{attribute 'linkalways'} 
{attribute 'no_explicit_call' := 'This FB is a CLASS and must be accessed using methods or properties'}
{attribute 'enable_dynamic_creation'}
FUNCTION_BLOCK Node_F_VN_FillContainerExp_INT EXTENDS VisionNode
VAR
    ipContainer : _ITcVnContainer;
    nValue : _INT(0);
    nStartIdx : _ULINT(0);
    nCount : _ULINT(0);
    hrPrev : _HRESULT(S_OK);
    hresult : _HRESULT(S_OK);
END_VAR

METHOD PUBLIC  Clone : I_Node
VAR
    pNode : POINTER TO Node_F_VN_FillContainerExp_INT;
END_VAR
pNode := __NEW(Node_F_VN_FillContainerExp_INT);
Clone := pNode^;
END_METHOD

METHOD FB_init : BOOL
VAR_INPUT
    bInitRetains : BOOL; // if TRUE, the retain variables are initialized (warm start / cold start)
    bInCopyCode : BOOL;  // if TRUE, the instance afterwards gets moved into the copy code (online change)
END_VAR
AddInput('ipContainer', ipContainer);
AddParameter('nValue', nValue);
AddParameter('nStartIdx', nStartIdx);
AddParameter('nCount', nCount);
AddInput('hrPrev', hrPrev);
AddOutput('ipContainer', ipContainer);
AddOutput('hresult',hresult);
END_METHOD

METHOD PROTECTED OnExecute
hresult.Value := F_VN_FillContainerExp_INT(
    ipContainer := ipContainer.Value,
    nValue := nValue.Value,
    nStartIdx := nStartIdx.Value,
    nCount := nCount.Value,
    hrPrev:= hrPrev.Value);
END_METHOD

METHOD PUBLIC PreExecutionCheck
VAR_INPUT
    Check : I_PreExecutionChecks;
END_VAR
Check.IsTrue(ipContainer.IsValid, 'ipContainer must be a valid container');
Check.IsTrue(ipContainer.IsType(TC_GLOBAL_CONST_LIST.ContainerType_Vector_INT), 'ipContainer contains incorrect type');
END_METHOD

END_FUNCTION_BLOCK

(* stored: Version 1.1.0.1, ProductVersion 3.1.4026.13
   POU Node_F_VN_FillContainerExp_INT: Id {23b78316-4d38-47ad-b72d-6bd99bc2952d}, SpecialFunc None
   Folder Constructor: Id {af9372ec-d9cd-43f4-8171-491f02b612e3}
   Method Clone: Id {80c76df1-6869-4f4d-bd88-ae6120653396}
   Method FB_init: Id {37b7e1e6-f4a0-4281-8250-03dfa2b30695}
   Method OnExecute: Id {b7b7c924-0465-4b5b-a04d-5ed4c74063ab}
   Method PreExecutionCheck: Id {18b8b318-b61a-4f48-a4e1-aae5302935e1} *)
